(* IEC 61131-3 sources: OpenPLC_Tutorials/Ladder Logic and Ladder Diagram/05 XOR and XNOR Gate/05 XOR and XNOR Gate/build, 2 files *)

(* ---- plc.st ---- *)
TYPE
  LOGLEVEL : (CRITICAL, WARNING, INFO, DEBUG) := INFO;
END_TYPE

FUNCTION_BLOCK LOGGER
  VAR_INPUT
    TRIG : BOOL;
    MSG : STRING;
    LEVEL : LOGLEVEL := INFO;
  END_VAR
  VAR
    TRIG0 : BOOL;
  END_VAR

  IF TRIG AND NOT TRIG0 THEN
  {{
   LogMessage(GetFbVar(LEVEL),(char*)GetFbVar(MSG, .body),GetFbVar(MSG, .len));
  }}
  END_IF;
  TRIG0:=TRIG;
END_FUNCTION_BLOCK

PROGRAM XOR_and_XNOR
  VAR
    INPUT_0 : BOOL;
    INPUT_1 : BOOL;
    INPUT_2 : BOOL;
    INPUT_3 : BOOL;
    OUTPUT_0 : BOOL;
    OUTPUT_1 : BOOL;
  END_VAR

  OUTPUT_0 := NOT(INPUT_0) AND INPUT_1 OR NOT(INPUT_1) AND INPUT_0;
  OUTPUT_1 := INPUT_3 AND INPUT_2 OR NOT(INPUT_3) AND NOT(INPUT_2);
END_PROGRAM

CONFIGURATION Config0

  RESOURCE Res0 ON PLC
    TASK task0(INTERVAL := T#20ms,PRIORITY := 0);
    PROGRAM instance0 WITH task0 : XOR_and_XNOR;
  END_RESOURCE
END_CONFIGURATION

(* ---- generated_plc.st ---- *)
PROGRAM XOR_and_XNOR
  VAR
    INPUT_0 : BOOL;
    INPUT_1 : BOOL;
    INPUT_2 : BOOL;
    INPUT_3 : BOOL;
    OUTPUT_0 : BOOL;
    OUTPUT_1 : BOOL;
  END_VAR

  OUTPUT_0 := NOT(INPUT_0) AND INPUT_1 OR NOT(INPUT_1) AND INPUT_0;
  OUTPUT_1 := INPUT_3 AND INPUT_2 OR NOT(INPUT_3) AND NOT(INPUT_2);
END_PROGRAM

CONFIGURATION Config0

  RESOURCE Res0 ON PLC
    TASK task0(INTERVAL := T#20ms,PRIORITY := 0);
    PROGRAM instance0 WITH task0 : XOR_and_XNOR;
  END_RESOURCE
END_CONFIGURATION
